PROGRAM PRG_INJ
VAR
END_VAR


// Valves
VCN_70(i_xExtIlkOK:= , i_ReqPos:= , iq_stVCN=> );
//VGP_80
VVC_71(i_xExtILK_OK:= VVC_72.M_IsClosed(), i_xOverrideMode:= , iq_stValve=> );
VVC_72(i_xExtILK_OK:= VVC_71.M_IsClosed(), i_xOverrideMode:= , iq_stValve=> );

//Gauges
GCM_70(PG=> , i_rFULL_SCALE:= 2000);
GCM_80(PG=> , i_rFULL_SCALE:= 20);
GCM_81(PG=> , i_rFULL_SCALE:= 0.25);
// Set bits for EL3174-0002
GCM_70.M_SetBits(30518);
GCM_80.M_SetBits(30518);
GCM_81.M_SetBits(30518);

END_PROGRAM

(* stored: Version 1.1.0.1, ProductVersion 3.1.4022.18
   POU PRG_INJ: Id {8b858f89-a705-4da6-a8c0-4cd0b412d38f}, SpecialFunc None *)
